Omron CX-Programmer project NewProject (CX-Programmer 9.50)

# PLC plc1: CJ2H CPU64

## Global symbols (name address type ; comment)
0.00 BOOL  ; On
0.01 BOOL  ; off
10.00 BOOL  ; lampu

## Program NewProgram1 (cyclic task 0)

### Section Section1

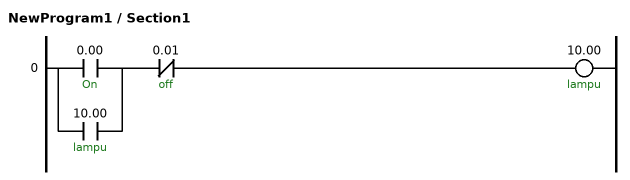
; rung 0
LD 0.00  ; On
OR 10.00  ; lampu
ANDNOT 0.01  ; off
OUT 10.00  ; lampu

### Section END
; rung 0
END(001)